FUNCTION_BLOCK FB_TestSystem EXTENDS FB_SystemContinous
VAR_INPUT
END_VAR
VAR_OUTPUT
END_VAR
VAR	
	//OPC UA structures
	{attribute 'OPC.UA.DA' := '1'}
	localSetParameters : ST_TestSystemSetParameters;
	{attribute 'OPC.UA.DA' := '1'}
	localState : ST_TestSystemState;	

	//default parameters
	localDefaultParameters : ST_TestSystemDefaultParameters;
	
	//digital input
	bOperational 				AT %I*: BOOL;
	
	//digital output
	bSystemOperationOn 			AT %Q*: BOOL := FALSE;
		
	//Components - Pump
	ST_PumpDefaultParameters : ST_GundfosMagna3DefaultParameters := (bExternalTemperatureSensor := TRUE,aSetPointLimitsConstantSpeed := [0,100]);
	pump			 			: FB_PumpGrundfosMagna3 := (ST_DefaultParameters := ST_PumpDefaultParameters); 
	bStartPump					: BOOL := FALSE;
	fSetPointPump 				: REAL := 50;
	bAlgorithmPermissionPump 	: BOOL := FALSE;
	nControlModePump : E_GrundfosMagna3ControlMode := 0;
	
	//Components - Discrete Valve
	ST_DiscreteValveDefaultParameters : ST_DiscreteValveDefaultParameters := (bFeedbackSignal := TRUE);
	discreteValve				: FB_DiscreteValve := (ST_DefaultParameters := ST_DiscreteValveDefaultParameters);
	bOpenValve					: BOOL := FALSE;
	
	//Components - Controlled Valve
	ST_ControledValveDefaultParameters : ST_MixingValveDefaultParameters := (bFeedbackSignal := TRUE, fControlerAmplification := 0.5, fControlerIntegralTime := 500);
	controledValve 					: FB_MixingValve := (ST_DefaultParameters := ST_ControledValveDefaultParameters);
	bOpenControledValve 				: BOOL := FALSE;
	fSetpointControledValve 			: REAL := 75;
	
	nInit						: BOOL := FALSE;
	

END_VAR

//set init values
IF(NOT nInit) THEN
	fSetPointAutomatic := 20;
	bAlgorithmPermission := TRUE;
	nInit := TRUE;
END_IF

//start system methods
MAIN();
SetState();//set state values

//pump
pump(
	bSetStatusOnAutomatic := bStartPump,
	fSetPointAutomatic := fSetPointPump,
	bAlgorithmPermission := bAlgorithmPermissionPump,
	nControlModeAutomatic := nControlModePump
);
pump.SetState_Profibus();

//discrete valve
discreteValve(
	bSetStatusOnAutomatic := bOpenValve,
	bAlgorithmPermission := bAlgorithmPermissionPump);
discreteValve.SetState_BI_BO();
	
//controlled valve
controledValve(
	bSetStatusOnAutomatic := bOpenControledValve,
	bAlgorithmPermission := bAlgorithmPermissionPump,
	fSetPointAutomatic := fSetpointControledValve);
controledValve.SetState_AI_AO();

METHOD PROTECTED  Operational : BOOL
VAR_INPUT
END_VAR
VAR_OUTPUT
	bSwitchToWorking : BOOL := FALSE;
END_VAR
bSystemOperationOn := TRUE;
bSwitchToWorking := TRUE;
END_METHOD

METHOD PROTECTED  RampDown : BOOL
VAR_INPUT
END_VAR
VAR_OUTPUT
	bRampDownFinished : BOOL := FALSE;
END_VAR
IF bOperational=FALSE THEN
	//turn pump off
	bStartPump := FALSE;
	fSetPointPump := 0;	
END_IF

IF bOperational=FALSE AND pump.controlState.bStatusOn=FALSE THEN
	bOpenValve := FALSE;
END_IF

IF bOperational=FALSE AND pump.controlState.bStatusOn=FALSE AND discreteValve.controlState.bStatusOn=FALSE THEN
	bRampDownFinished := TRUE;
END_IF
END_METHOD

METHOD PROTECTED  RampUp : BOOL
VAR_INPUT
END_VAR
VAR_OUTPUT
	bRampUpFinished : BOOL := FALSE;
END_VAR
VAR
END_VAR
//open valves
bOpenValve := TRUE;
bOpenControledValve := TRUE;

//turn pump on
bStartPump := TRUE;
fSetPointPump := 60.00;

IF pump.bStatusOn = TRUE THEN
	bRampUpFinished := TRUE;
END_IF;
END_METHOD

METHOD PROTECTED   SetSetPointLimits : BOOL
VAR_INPUT
END_VAR
aSetPointLimits := localDefaultParameters.aSetPointLimits;
END_METHOD

METHOD PROTECTED   SetState : BOOL
VAR_INPUT
END_VAR
//copy states to OPC UA
controlState.bStatusOn := bSystemOperationOn;

//set outputs from OPC UA
bSystemOperationOn := localSetParameters.bSystemOperationOn;
END_METHOD

METHOD PROTECTED  StateCheck : BOOL
(* In this method the folowing elements of the actorState structrure have to be set if they are not set yet:
	bStatusOn 		: BOOL; //status on / off
	bError			: BOOL; //true if in error
	sErrorMessage	: STRING; //returns error message
	bWarning		: BOOL; //true if in warning
	sWarningMessage	: STRING; //returns warning message
	fOperatingPoint	: REAL; //current operating point
*)
VAR_INPUT
END_VAR
VAR
END_VAR
END_METHOD

METHOD PROTECTED  Working : BOOL
VAR_INPUT
END_VAR
VAR_OUTPUT
	bSwitchToOperational : BOOL := FALSE;
END_VAR
//turn system off, e.g. according to hysteresis
//bSystemOperationOn := FALSE;
END_METHOD

END_FUNCTION_BLOCK

(* stored: Version 1.1.0.1, ProductVersion 3.1.4024.9
   POU FB_TestSystem: Id {7003cb31-5239-49d6-8372-83a96f9671f9}, SpecialFunc None
   Method Operational: Id {f0511b9d-ec63-4439-bedf-00ea55360bc5}
   Method RampDown: Id {b7b74ab3-d092-435e-8cae-255bb8b32b0c}
   Method RampUp: Id {f3784821-29fa-4a43-84ee-d8fad2aad1d8}
   Method SetSetPointLimits: Id {f051f01d-b197-4bf8-82e6-ce2ab19a0807}
   Method SetState: Id {6f5b6a90-4211-4d68-92aa-fa3fb40b781b}
   Method StateCheck: Id {d5772649-a060-4f63-863c-5518172c4e38}
   Method Working: Id {108f57c1-42ce-4e97-b194-08b3f4031db8} *)
